SUBAPPLICATION OuterSubApp (* Subapplication Type *)
  (* Standard: 61499-2 *)
  (* Version 1.0, 2024-08-05, mario *)
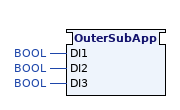
  VAR_INPUT
    DI1 : BOOL := TRUE;
    DI2 : BOOL := FALSE;
    DI3 : BOOL := TRUE;
  END_VAR
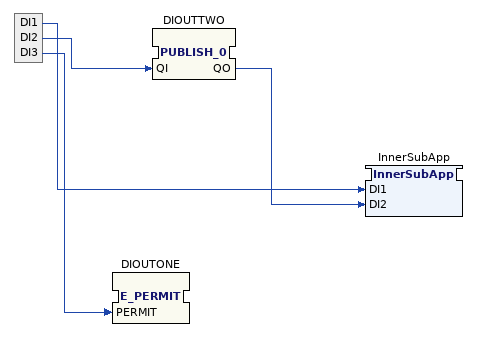
  FBS
    DIOUTONE : E_PERMIT;
    DIOUTTWO : PUBLISH_0;
  END_FBS
  SUBAPPS
    InnerSubApp : InnerSubApp;
  END_SUBAPPS
  DATA_CONNECTIONS
    DI1 TO InnerSubApp.DI1;
    DI3 TO DIOUTONE.PERMIT;
    DI2 TO DIOUTTWO.QI;
    DIOUTTWO.QO TO InnerSubApp.DI2;
  END_CONNECTIONS
END_SUBAPPLICATION
